// Mitsubishi GX Works2 project: PLC_PART_B_GROUP7   PLC: FX3U/FX3UC

// global labels: Global1
VAR_GLOBAL
  start_machine AT X007 : BOOL;
  sent_temp20 AT X000 : BOOL;
  sen_temp10 AT X001 : BOOL;
  print_button AT X005 : BOOL;
  is_color AT X002 : BOOL;
  is_alarm AT X003 : BOOL;
  Light_fan AT Y001 : BOOL;
  Light_problem AT Y003 : BOOL;
  help_light_print AT M0 : BOOL;
  Timer_problem AT TC1 : BOOL;
  Timer_problem_state AT TS1 : BOOL;
  help_light_problem AT M1 : BOOL;
END_VAR
VAR_GLOBAL CONSTANT
  Timer_problem_dur : INT := 5;
  Timer_printing_time : INT := 25;
END_VAR
VAR_GLOBAL
  Light_print1 AT Y004 : BOOL;
  Light_print2 AT Y005 : BOOL;
  Timer_print AT TC2 : BOOL;
  temp AT D1100 : INT;
  Timer_print_state AT TS2 : BOOL;
  help_light_state AT M2 : BOOL;
  Light_alternate1 AT TC3 : BOOL;
  Light_alternate_state AT TS3 : BOOL;
  Light_alternate2 AT TC4 : BOOL;
  Light_alternate_state2 AT TS4 : BOOL;
  help_system_on AT M3 : BOOL;
  Light_system AT Y000 : BOOL;
  System_close AT X006 : BOOL;
END_VAR

// task Task_01 (event TRUE, interval 0, priority 31): POU_01

PROGRAM POU_01
(* structured ladder/FBD written out as ST: instructions are called as NAME(EN, inputs, outputs); _pN, _eN, _tN stand for wires *)
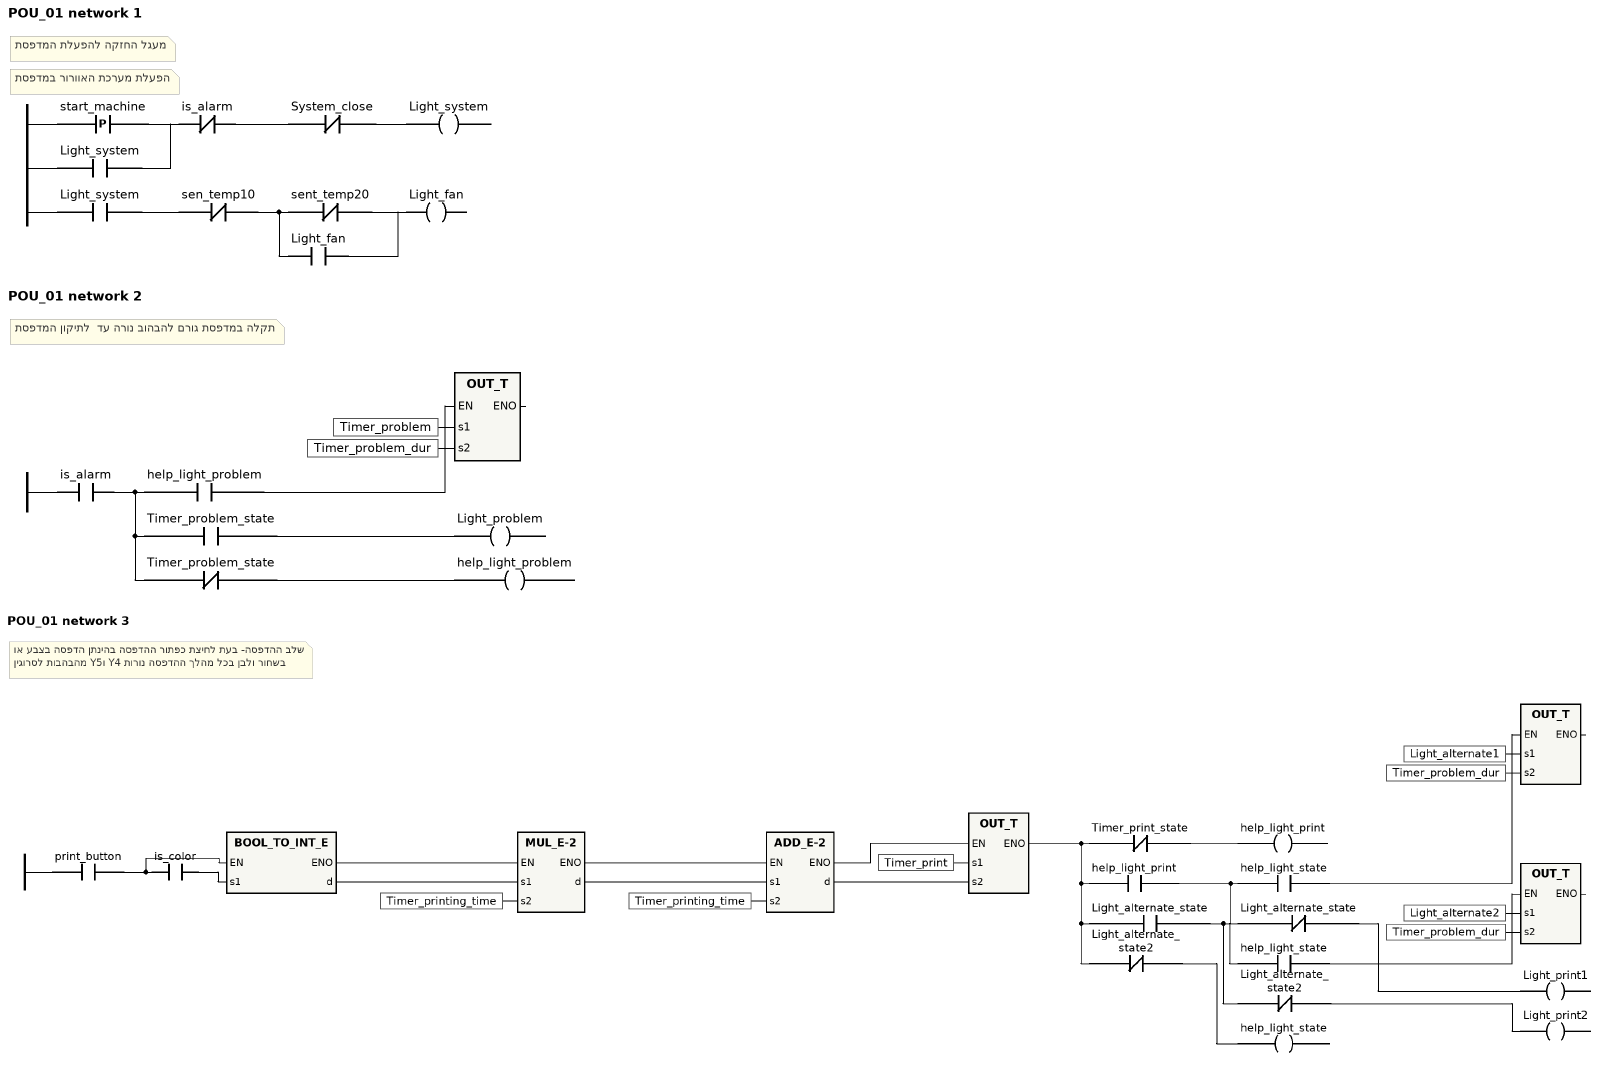
(* network 1 *)
(* מעגל החזקה להפעלת המדפסת *)
(* הפעלת מערכת האוורור במדפסת *)
Light_system := ((LDP(TRUE, start_machine) OR Light_system) AND NOT is_alarm) AND NOT System_close;
_p1 := Light_system AND NOT sen_temp10;
Light_fan := (_p1 AND NOT sent_temp20) OR (_p1 AND Light_fan);
(* network 2 *)
(* תקלה במדפסת גורם להבהוב נורה עד  לתיקון המדפסת *)
OUT_T(is_alarm AND help_light_problem, Timer_problem, Timer_problem_dur);
Light_problem := is_alarm AND Timer_problem_state;
help_light_problem := is_alarm AND NOT Timer_problem_state;
(* network 3 *)
(* שלב ההדפסה- בעת לחיצת כפתור ההדפסה בהינתן הדפסה בצבע או בשחור ולבן בכל מהלך ההדפסה נורות Y4 וY5 מהבהבות לסרוגין *)
_e2 := BOOL_TO_INT_E(print_button, print_button AND is_color, _t1);
_e4 := MUL_E(_e2, _t1, Timer_printing_time, _t3);
_e6 := ADD_E(_e4, _t3, Timer_printing_time, _t5);
_e7 := OUT_T(_e6, Timer_print, _t5);
help_light_print := _e7 AND NOT Timer_print_state;
_p8 := _e7 AND help_light_print;
OUT_T(_p8 AND help_light_state, Light_alternate1, Timer_problem_dur);
Light_print1 := _p8 AND NOT Light_alternate_state;
_p9 := _e7 AND Light_alternate_state;
OUT_T(_p9 AND help_light_state, Light_alternate2, Timer_problem_dur);
Light_print2 := _p9 AND NOT Light_alternate_state2;
help_light_state := _e7 AND NOT Light_alternate_state2;
END_PROGRAM
